TYPE ST_DetectDiameterStatus EXTENDS ST_StatusBasic :
STRUCT
	AllowGetPhoto : BOOL;
END_STRUCT
END_TYPE

(* stored: Version 1.1.0.1, ProductVersion 3.1.4024.13
   DUT ST_DetectDiameterStatus: Id {110821e3-dc89-48aa-9c70-b57ef9cb8f36} *)
